FUNCTION_BLOCK OUT_QO_US (* Combined display of QO & UINT STATUS outputs with event notification *)
  (* Standard: 61499-1; Classification: HMI; Function: Output; Type: QO + UINT STATUS *)
  (* Version 0.0, 2007-12-25, JHC, Holobloc Inc *)
  (* Compiler header: package fb.rt.hmi; *)
  (* Compiler Java Sun JDK 1.6.0 *)
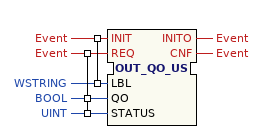
  EVENT_INPUT
    INIT WITH LBL; (* Initialization Request *)
    REQ WITH QO, STATUS; (* Normal Execution Request *)
  END_EVENT
  EVENT_OUTPUT
    INITO; (* Initialization Confirm *)
    CNF; (* Execution Confirmation *)
  END_EVENT
  VAR_INPUT
    LBL : WSTRING; (* Label to be displayed in leftmost field, next to event notification output *)
    QO : BOOL; (* QO value to be displayed *)
    STATUS : UINT;
  END_VAR
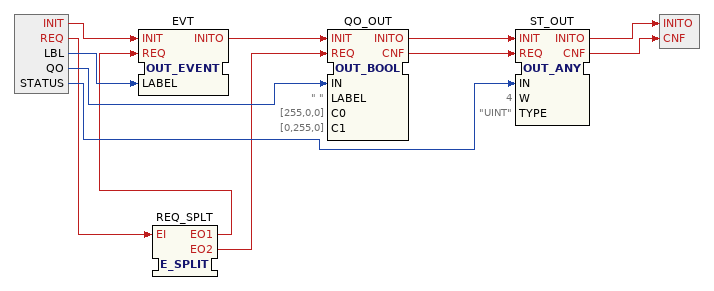
  FBS
    EVT : OUT_EVENT; (* Event notification display with main label (LBL) *)
    QO_OUT : OUT_BOOL(LABEL := "   ", C0 := [255,0,0], C1 := [0,255,0]);
    ST_OUT : OUT_ANY(W := 4, TYPE := "UINT");
    REQ_SPLT : E_SPLIT;
  END_FBS
  EVENT_CONNECTIONS
    INIT TO EVT.INIT;
    EVT.INITO TO QO_OUT.INIT;
    QO_OUT.INITO TO ST_OUT.INIT;
    QO_OUT.CNF TO ST_OUT.REQ;
    ST_OUT.INITO TO INITO;
    ST_OUT.CNF TO CNF;
    REQ TO REQ_SPLT.EI;
    REQ_SPLT.EO1 TO EVT.REQ;
    REQ_SPLT.EO2 TO QO_OUT.REQ;
  END_CONNECTIONS
  DATA_CONNECTIONS
    LBL TO EVT.LABEL;
    QO TO QO_OUT.IN;
    STATUS TO ST_OUT.IN;
  END_CONNECTIONS
END_FUNCTION_BLOCK
